(* PLC project MTPModule, Beckhoff Automation GmbH TwinCAT PLC Control 3.5.20.60 *)
(* stored: creationDateTime 2025-09-14T09:18:47.0031185, modificationDateTime 2025-09-14T09:18:47.0031185 *)

(* ************************************************************************ * This file was automatically generated by TwinCAT 3 MTP Engineering. * * * * INFO: This function block was generated for the possibility of * * using custom PID logic. See documentation for further details. * * * * Generated on: 9/10/2025 7:49:53 PM * * TwinCAT 3 MTP Engineering Version: 0.9.19.0 * ************************************************************************ *)
FUNCTION_BLOCK FB_MTP_PIDCtrl EXTENDS FB_MTP_PIDCtrlBase
  VAR
    CTRL_PID : FB_CTRL_PID;  (* Controller Toolbox (delete if you want to use own PID Logic) *)
    PIDParams : ST_Ctrl_PID_PARAMS;
    reset : BOOL;  (* Command to reset the PID controller, needed to reset errors *)
    counter : INT;
    errorID : INT;
    error : BOOL;
    hold : BOOL;
  END_VAR

            PIDLogic();
          

METHOD PROTECTED PIDLogic : BOOL
                  

// TODO: temporary bug fix: force auto mode:
StateAutAct := TRUE;
StateOffAct := FALSE;
StateOpAct := FALSE;

// reset the PID Controller
// (for example needed when there is an error)
IF reset THEN
	// trigger the reset method
	ResetPID();
	// reset the reset command
	reset := FALSE;
END_IF

// Set PID Params
PIDParams.tCtrlCycleTime	:= LREAL_TO_TIME(fCycleTime * 1000); // fCycleTime
PIDParams.tTaskCycleTime	:= LREAL_TO_TIME(fCycleTime * 1000);
PIDParams.fKp				:= P;
PIDParams.tTn				:= REAL_TO_TIME(TI * 1000);
PIDParams.tTv				:= REAL_TO_TIME(TD * 1000);
PIDParams.fOutMaxLimit		:= MVMax;
PIDParams.fOutMinLimit		:= MVMin;
PIDParams.bARWOnIPartOnly	:= TRUE;

PIDParams.bPInTheFeedbackPath := TRUE;

// Call Controller Toolbox PID function block
CTRL_PID(
	fSetpointValue:= SP,
	fActualValue:= PV,
	fManSyncValue:= ,
	bSync:= ,
	eMode:= eCTRL_MODE_ACTIVE,
	bHold:= ,
	fOut => ,
	bARWactive => ,
	eState => ,
	eErrorId => ,
	bError => ,
	stParams:= PIDParams);

// Write resulting Manipulated Value to MTP function block
counter := counter + 1;
MV:= LREAL_TO_REAL(CTRL_PID.fOut);
errorID:= CTRL_PID.eErrorId;
error := CTRL_PID.bError;
hold := CTRL_PID.bHold;
                
END_METHOD

METHOD ResetPID : BOOL
                  // Reset PID
CTRL_PID(
	eMode := eCTRL_MODE_Reset,
	stParams:= PIDParams
);

// Write resulting Manipulated Value to MTP function block
MV:= LREAL_TO_REAL(CTRL_PID.fOut);
                
END_METHOD

(* FB_Init is always available implicitly and it is used primarily for initialization. The return value is not evaluated. For a specific influence, you can also declare the methods explicitly and provide additional code there with the standard initialization code. You can evaluate the return value. *)
METHOD FB_INIT : BOOL
  VAR_INPUT
    bInitRetains : BOOL;  (* TRUE: the retain variables are initialized (reset warm / reset cold) *)
    bInCopyCode : BOOL;  (* TRUE: the instance will be copied to the copy code afterward (online change) *)
  END_VAR
                  fCycleTime:= 1;
                
END_METHOD
END_FUNCTION_BLOCK
